FUNCTION_BLOCK TIMER
VAR_INPUT
	bStart : BOOL := TRUE;
END_VAR
VAR_OUTPUT
	tDifference : TIME;
END_VAR
VAR
	tTimeReturn1:	TIME;
	tTimeReturn2:	TIME;
	fbTrigger1:		R_TRIG;
	fbTrigger2:		F_TRIG;
END_VAR

fbTrigger1(CLK := bStart);
fbTrigger2(CLK := bStart);

IF fbTrigger1.Q THEN
	tTimeReturn1 := TIME();
END_IF

IF bStart OR fbTrigger2.Q THEN
	tTimeReturn2 := TIME();
END_IF

tDifference := tTimeReturn2 - tTimeReturn1;

END_FUNCTION_BLOCK

(* stored: Version 1.1.0.1, ProductVersion 3.1.4024.9
   POU TIMER: Id {7a6416e5-cc61-4d14-8bf3-453395375baf}, SpecialFunc None *)
